{attribute 'pack_mode' := '1'}
    {attribute 'OPC.UA.DA' := '1'}
    {attribute 'OPC.UA.DA.StructuredType' := '1'}
    (*
    ST_RW_IntMb_HMI_IgnitionExp
    ==================================================
    Generated from Ignition UDT: RW_Int_MB
    Total tags: 1
    Generated on: 2025-09-12 15:49:02
    *)
    TYPE ST_RW_IntMb_HMI_IgnitionExp :
    STRUCT
        {attribute 'OPC.UA.DA' := '1'}
        {attribute 'OPC.UA.DA.Description' := '{Description}'}
        // {Description}
        Value : DINT := 0;
    END_STRUCT
    END_TYPE

(* stored: Version 1.1.0.1
   DUT ST_RW_IntMb_HMI_IgnitionExp: Id {1465de4e-0261-46e0-a284-58a0ce961720} *)
